FUNCTION_BLOCK FB_LiftA_Extended EXTENDS FB_Lift
// This is an extended functionblock of FB_Lift. This Functionblock is for Lift A (Depalletizer)
VAR_INPUT

END_VAR
VAR_OUTPUT
	o_xTaskDone : BOOL;
END_VAR
VAR	
	aLayerHeights	: ARRAY[1..10] OF INT;
END_VAR

iConveyorHeight := 0;

CASE i_eMode OF
	eModus.Auto :
	CASE i_eState OF
		eSingleState.Execute :
			CASE i_eLiftState OF
				eLiftStates.WaitForPallet :
					// Let a new pallet through if there are any.
					THIS^.WaitForPallet();
					
				eLiftStates.MoveUpToLayer :
				 	// Go to the next layer.
					THIS^.MoveUpToLayer();

				eLiftStates.CheckNextLayer :
					// Check if it is possible to move up.
					THIS^.CheckNextLayer();
					
			END_CASE
	END_CASE
	
	eModus.Manual :
		// Doe effe zelf																			// TOEVOEGEN MET HMI
		// Lift handmatig bedienen door INT invoer?
		// Pins handmatig in en uit, met beveiliging zodat pallet niet naar beneden dondert
	eModus.Off :
		// Doe niks
		// Stop
END_CASE

METHOD CheckNextLayer : BOOL
VAR_INPUT
	
END_VAR

VAR

END_VAR
// Nog maken
END_METHOD

METHOD MoveUpToLayer : BOOL
VAR_INPUT
END_VAR
END_METHOD

METHOD WaitForPallet : BOOL
VAR_INPUT
	
END_VAR

VAR
	fbKlep : FB_Klep;
END_VAR
// Wanneer in Normal Height positie, laat pallet door.
// Check welke lift het is. Dan uitvoeren wat voor dat deel werkt.
o_xNewPalletPossible := TRUE; // Command to start conveyor

IF i_xLightSensor1 AND NOT i_xLightSensor2 THEN
//Klep omhoog														TOEVOEGEN
	fbKlep(i_eAutoWantedPosition := 1);
END_IF

IF NOT i_xLightSensor1 AND i_xLightSensor2 THEN
o_xNewPalletPossible := FALSE; // Stop conveyor
o_xPalletInPosition := TRUE;
END_IF

IF o_xPalletInPosition THEN
i_eLiftState := eLiftStates.Impale;
END_IF
END_METHOD

END_FUNCTION_BLOCK

(* stored: Version 1.1.0.1
   POU FB_LiftA_Extended: Id {29ce4f32-d5ec-44c6-b550-ed18c3714c4b}, SpecialFunc None
   Method CheckNextLayer: Id {8f1d2526-a33e-4d40-9997-1757c01d0527}
   Method MoveUpToLayer: Id {3339177a-337e-4fd8-a5b4-139eb710ec0a}
   Method WaitForPallet: Id {411af908-da43-45f2-beac-587db957c43f} *)
